Fanuc KAREL source: kt00491.KL

-- PROVISIONAL review KL for V1013-1; original PC SHA256 af34c7b7e4d4474d170201845d7764e7a265961c47999d9139edc78af9ec86bb
-- Incomplete behavior may be omitted. Consult companion uncertainty JSON. Do not deploy.
PROGRAM KT00491
%NOLOCKGROUP
-- UNRESOLVED_DECL P1 type=000101
-- UNRESOLVED_DECL P2 type=000199
-- UNRESOLVED_DECL OUT type=000106
BEGIN
  -- UNRESOLVED_PC offsets 5-39; opcodes 49,49,7E,60,7E,4A
  -- UNRESOLVED_PC offsets 44-48; opcodes 7F
END KT00491
